// Mitsubishi GX Works2 project: TramCapPhoiAuto   PLC: FX2N/FX2NC

PROGRAM MAIN
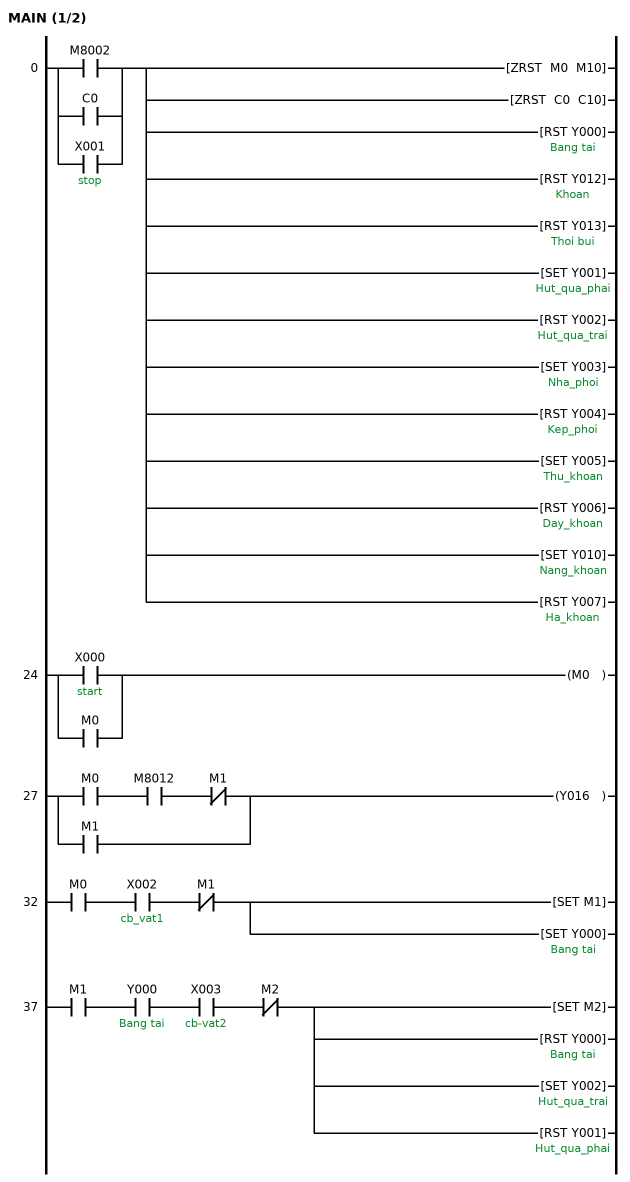
0     LD      M8002
      OR      C0
      OR      X001  ; stop
      ZRST    M0 M10
      ZRST    C0 C10
      RST     Y000  ; Bang tai
      RST     Y012  ; Khoan
      RST     Y013  ; Thoi bui
      SET     Y001  ; Hut_qua_phai
      RST     Y002  ; Hut_qua_trai
      SET     Y003  ; Nha_phoi
      RST     Y004  ; Kep_phoi
      SET     Y005  ; Thu_khoan
      RST     Y006  ; Day_khoan
      SET     Y010  ; Nang_khoan
      RST     Y007  ; Ha_khoan
24    LD      X000  ; start
      OR      M0
      OUT     M0
27    LD      M0
      AND     M8012
      ANI     M1
      OR      M1
      OUT     Y016
32    LD      M0
      AND     X002  ; cb_vat1
      ANI     M1
      SET     M1
      SET     Y000  ; Bang tai
37    LD      M1
      AND     Y000  ; Bang tai
      AND     X003  ; cb-vat2
      ANI     M2
      SET     M2
      RST     Y000  ; Bang tai
      SET     Y002  ; Hut_qua_trai
      RST     Y001  ; Hut_qua_phai
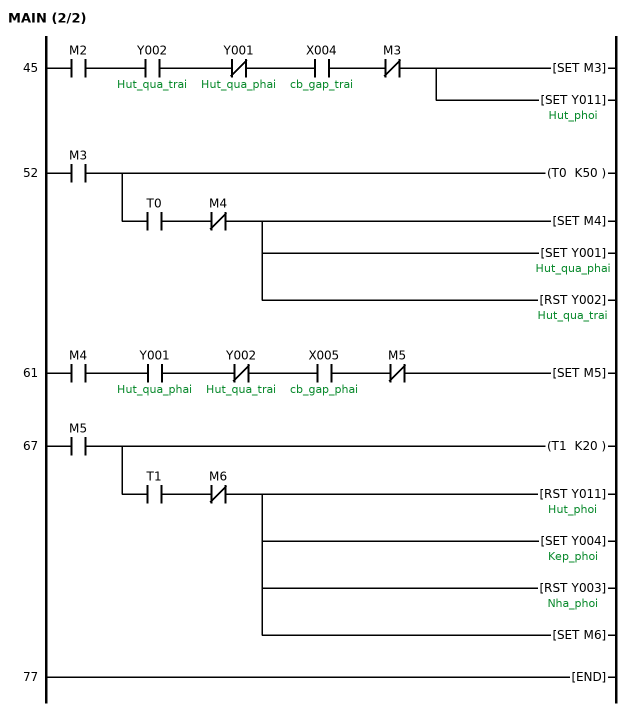
45    LD      M2
      AND     Y002  ; Hut_qua_trai
      ANI     Y001  ; Hut_qua_phai
      AND     X004  ; cb_gap_trai
      ANI     M3
      SET     M3
      SET     Y011  ; Hut_phoi
52    LD      M3
      OUT     T0 K50
      AND     T0
      ANI     M4
      SET     M4
      SET     Y001  ; Hut_qua_phai
      RST     Y002  ; Hut_qua_trai
61    LD      M4
      AND     Y001  ; Hut_qua_phai
      ANI     Y002  ; Hut_qua_trai
      AND     X005  ; cb_gap_phai
      ANI     M5
      SET     M5
67    LD      M5
      OUT     T1 K20
      AND     T1
      ANI     M6
      RST     Y011  ; Hut_phoi
      SET     Y004  ; Kep_phoi
      RST     Y003  ; Nha_phoi
      SET     M6
77    END
END_PROGRAM

// device comments not shown above
X007  ; cb_giu_trong
X010  ; cb_giu_ngoai
X011  ; cb_day_khoan
X012  ; cb_thu_khoan
X013  ; cb_ha_khoan
X014  ; cb_nang_khoan
